FUNCTION_BLOCK FB_SituarPale_SFC_1
VAR_INPUT
	//nuestras_variables
	Tcinta: TIME := T#0.5S;

	
    // SFC-Flags
    SFCPause: BOOL;
    SFCReset: BOOL;
    
    // Indicadores de sincronizacion
    Ack: BOOL := TRUE;
    Execute: BOOL;
	
	//Entradas
   	Presencia_pale: BOOL;
	Vertical_descargador_abajo: BOOL;
	Vacio_obtenido_vacuostato_descargador: BOOL;
	Vertical_descargador_arriba: BOOL;
	Horizontal_descargador_delante: BOOL;
	Vertical_descargador_arriba: BOOL;
	
END_VAR
VAR_OUTPUT
    // Indicadores de sincronizacion
    Done: BOOL;
    Ready: BOOL;

	//Salidas
	Activa_marcha_motor_cinta: BOOL;
END_VAR
VAR
END_VAR

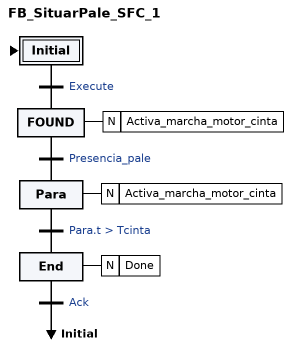
INITIAL_STEP Initial:
END_STEP
TRANSITION FROM Initial TO FOUND
    := Execute;
END_TRANSITION
STEP FOUND:
    Activa_marcha_motor_cinta(N);
END_STEP
TRANSITION FROM FOUND TO Para
    := Presencia_pale;
END_TRANSITION
STEP Para:
    Activa_marcha_motor_cinta(N);
END_STEP
TRANSITION FROM Para TO End
    := Para.t > Tcinta;
END_TRANSITION
STEP End:
    Done(N);
END_STEP
TRANSITION FROM End TO Initial
    := Ack;
END_TRANSITION

END_FUNCTION_BLOCK

(* stored: Version 1.1.0.1, ProductVersion 3.1.4024.12
   POU FB_SituarPale_SFC_1: Id {273a3972-5d8d-433a-b32e-61ca959a9370}, SpecialFunc None *)
